TYPE EL3052_HWTOPLC_PDOS :
	STRUCT
		
	
	Channel1 	AT %I* : EL3052_CHANNEL;
	Channel2 	AT %I* : EL3052_CHANNEL;



	END_STRUCT
END_TYPE

(* stored: Version 1.1.0.1, ProductVersion 3.1.4024.15
   DUT EL3052_HWTOPLC_PDOS: Id {66d94412-8d8d-47bb-a0b0-55a9c586f39f} *)
